(* PLC project Desconhecido, UFSCar Conversor PNML2Ladder 1 *)
(* stored: creationDateTime 2025-01-15T12:13:14, modificationDateTime 2025-02-12T16:11:11 *)

PROGRAM instance0

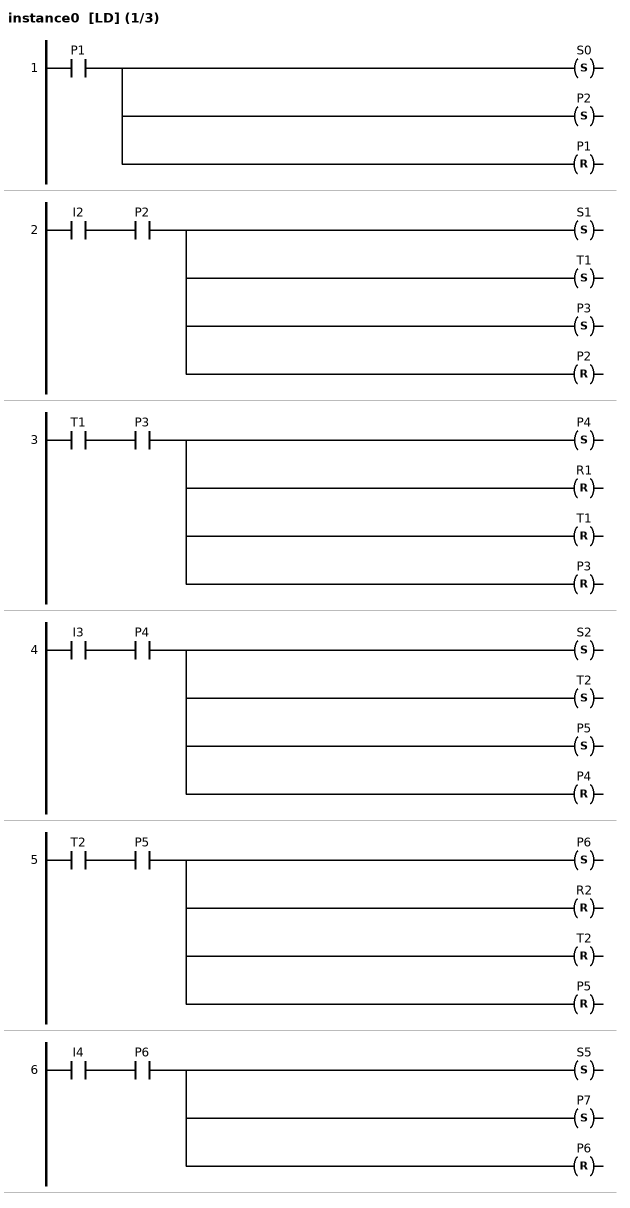
(* LD diagram, written out as Structured Text *)
IF P1 THEN S0 := TRUE; END_IF;
IF P1 THEN P2 := TRUE; END_IF;
IF P1 THEN P1 := FALSE; END_IF;
IF I2 AND P2 THEN S1 := TRUE; END_IF;
IF I2 AND P2 THEN T1 := TRUE; END_IF;
IF I2 AND P2 THEN P3 := TRUE; END_IF;
IF I2 AND P2 THEN P2 := FALSE; END_IF;
IF T1 AND P3 THEN P4 := TRUE; END_IF;
IF T1 AND P3 THEN R1 := FALSE; END_IF;
IF T1 AND P3 THEN T1 := FALSE; END_IF;
IF T1 AND P3 THEN P3 := FALSE; END_IF;
IF I3 AND P4 THEN S2 := TRUE; END_IF;
IF I3 AND P4 THEN T2 := TRUE; END_IF;
IF I3 AND P4 THEN P5 := TRUE; END_IF;
IF I3 AND P4 THEN P4 := FALSE; END_IF;
IF T2 AND P5 THEN P6 := TRUE; END_IF;
IF T2 AND P5 THEN R2 := FALSE; END_IF;
IF T2 AND P5 THEN T2 := FALSE; END_IF;
IF T2 AND P5 THEN P5 := FALSE; END_IF;
IF I4 AND P6 THEN S5 := TRUE; END_IF;
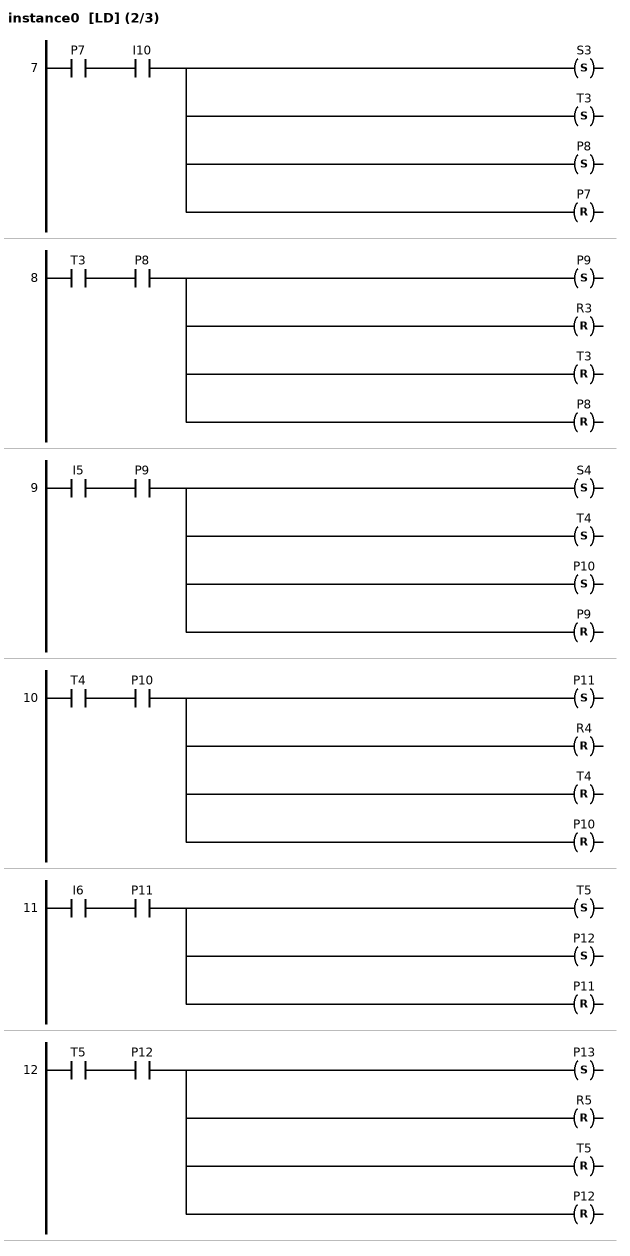
IF I4 AND P6 THEN P7 := TRUE; END_IF;
IF I4 AND P6 THEN P6 := FALSE; END_IF;
IF P7 AND I10 THEN S3 := TRUE; END_IF;
IF P7 AND I10 THEN T3 := TRUE; END_IF;
IF P7 AND I10 THEN P8 := TRUE; END_IF;
IF P7 AND I10 THEN P7 := FALSE; END_IF;
IF T3 AND P8 THEN P9 := TRUE; END_IF;
IF T3 AND P8 THEN R3 := FALSE; END_IF;
IF T3 AND P8 THEN T3 := FALSE; END_IF;
IF T3 AND P8 THEN P8 := FALSE; END_IF;
IF I5 AND P9 THEN S4 := TRUE; END_IF;
IF I5 AND P9 THEN T4 := TRUE; END_IF;
IF I5 AND P9 THEN P10 := TRUE; END_IF;
IF I5 AND P9 THEN P9 := FALSE; END_IF;
IF T4 AND P10 THEN P11 := TRUE; END_IF;
IF T4 AND P10 THEN R4 := FALSE; END_IF;
IF T4 AND P10 THEN T4 := FALSE; END_IF;
IF T4 AND P10 THEN P10 := FALSE; END_IF;
IF I6 AND P11 THEN T5 := TRUE; END_IF;
IF I6 AND P11 THEN P12 := TRUE; END_IF;
IF I6 AND P11 THEN P11 := FALSE; END_IF;
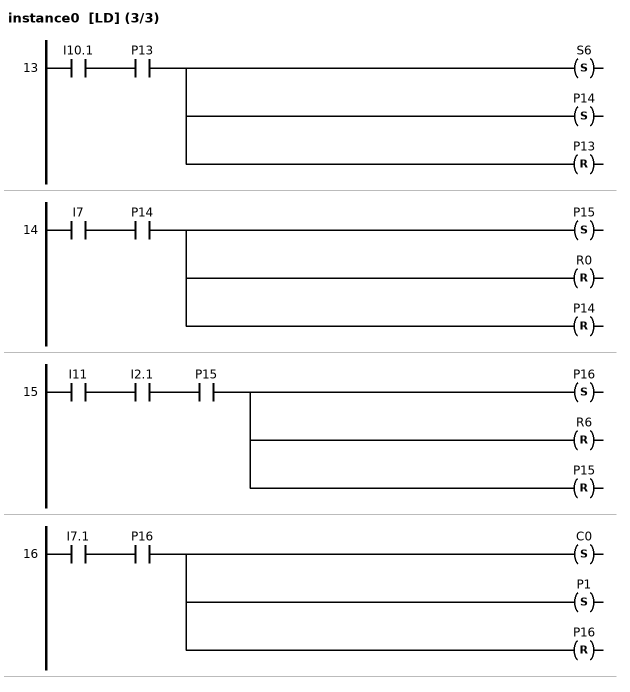
IF T5 AND P12 THEN P13 := TRUE; END_IF;
IF T5 AND P12 THEN R5 := FALSE; END_IF;
IF T5 AND P12 THEN T5 := FALSE; END_IF;
IF T5 AND P12 THEN P12 := FALSE; END_IF;
IF I10.1 AND P13 THEN S6 := TRUE; END_IF;
IF I10.1 AND P13 THEN P14 := TRUE; END_IF;
IF I10.1 AND P13 THEN P13 := FALSE; END_IF;
IF I7 AND P14 THEN P15 := TRUE; END_IF;
IF I7 AND P14 THEN R0 := FALSE; END_IF;
IF I7 AND P14 THEN P14 := FALSE; END_IF;
IF I11 AND I2.1 AND P15 THEN P16 := TRUE; END_IF;
IF I11 AND I2.1 AND P15 THEN R6 := FALSE; END_IF;
IF I11 AND I2.1 AND P15 THEN P15 := FALSE; END_IF;
IF I7.1 AND P16 THEN C0 := TRUE; END_IF;
IF I7.1 AND P16 THEN P1 := TRUE; END_IF;
IF I7.1 AND P16 THEN P16 := FALSE; END_IF;
END_PROGRAM

CONFIGURATION config0
  RESOURCE resource1 ON PLC
    TASK task0(INTERVAL := T#20ms, PRIORITY := 0);
    PROGRAM instance0 WITH task0 : program0;
  END_RESOURCE
END_CONFIGURATION
